KUKA KRL program: Dynamic_Mov.src

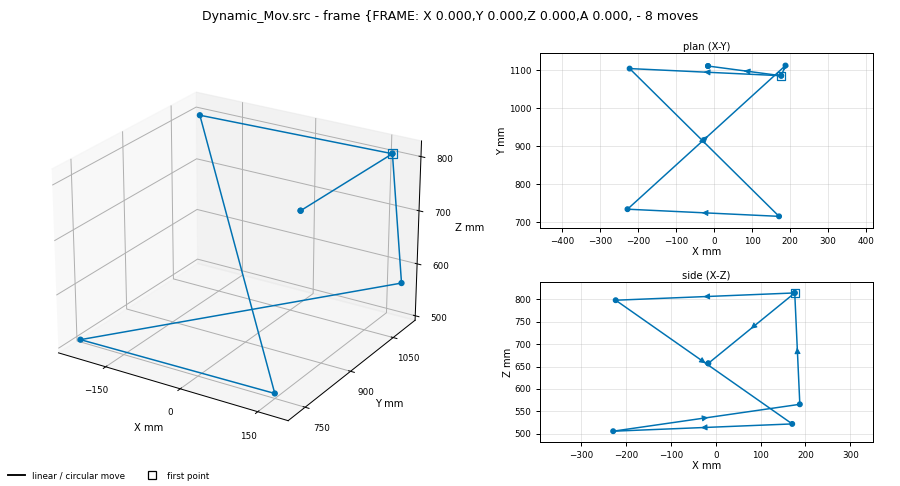
[picture p0: tool path of Dynamic_Mov.src in frame {FRAME: X 0.000,Y 0.000,Z 0.000,A 0.000,, 8 of 9 moves have a stored position in this frame; points joined in program order, loops and branches not executed]
&ACCESS RVP
&REL 1
&PARAM TEMPLATE = C:\KRC\Roboter\Template\vorgabe
&PARAM EDITMASK = *
DEF Kuka_Relative_Mo ( )
EXT BAS (BAS_COMMAND :IN,REAL :IN )


; GLOBAL INTERRUPT DECL 3 WHEN $STOPMESS==TRUE DO IR_STOPM ( )
; INTERRUPT ON 3

;FOLD Initialise and set default speed
BAS (#INITMOV,0)
BAS (#VEL_PTP,100)
BAS (#ACC_PTP,20)
$VEL.CP=0.2
BAS (#TOOL,0)
BAS (#BASE,0)
;ENDFOLD

;;FOLD STARTPOS
;$BWDSTART = FALSE
;PDAT_ACT = PDEFAULT
;BAS(#PTP_DAT)
;FDAT_ACT = {TOOL_NO 0,BASE_NO 0,IPO_FRAME #BASE}
;BAS(#FRAMES)
;;ENDFOLD

$ADVANCE = 5

;FOLD ---- Quickly skip BCO ----
; PTP $AXIS_ACT
;ENDFOLD

;FOLD ---- GO HOME ----
; PTP {A1 0.000, A2 -90.000, A3 90.000, A4 0.000, A5 0.000, A6 0.000, E1 0, E2 0, E3 0, E4 0, E5 0, E6 0}
;ENDFOLD


; Program generated by RoboDK v5.6.0 for KUKA KR 16 2 on 31/10/2023 10:24:52
; ---- Setting reference (Base) ----
$BASE = {FRAME: X 0.000,Y 0.000,Z 0.000,A 0.000,B 0.000,C 0.000}
; --------------------------
; ---- Setting tool (TCP) ----
; TOOL_DATA[1] = {FRAME: X 0.000,Y 0.000,Z 10.000,A 0.000,B 0.000,C 0.000}
$TOOL = {FRAME: X 0.000,Y 0.000,Z 10.000,A 0.000,B 0.000,C 0.000}
; $TOOL = TOOL_DATA[1]
; --------------------------
PTP {A1 -91.44,A2 -55.82,A3 116.05,A4 -4.21,A5 -66.58,A6 4.44}
; ---- Setting reference (Base) ----
$BASE = {FRAME: X 0.000,Y 0.000,Z 0.000,A 0.000,B 0.000,C 0.000}
; --------------------------
; ---- Setting tool (TCP) ----
$TOOL = {FRAME: X 0.000,Y 0.000,Z 10.000,A 0.000,B 0.000,C 0.000}
; --------------------------
LIN {X 176.195,Y 1085.310,Z 814.055,A 67.080,B 83.301,C -20.346}
; ---- Setting reference (Base) ----
$BASE = {FRAME: X 0.000,Y 0.000,Z 0.000,A 0.000,B 0.000,C 0.000}
; --------------------------
; ---- Setting tool (TCP) ----
$TOOL = {FRAME: X 0.000,Y 0.000,Z 10.000,A 0.000,B 0.000,C 0.000}
; --------------------------
LIN {X -223.032,Y 1104.150,Z 797.831,A 67.080,B 83.301,C -20.346}
; ---- Setting reference (Base) ----
$BASE = {FRAME: X 0.000,Y 0.000,Z 0.000,A 0.000,B 0.000,C 0.000}
; --------------------------
; ---- Setting tool (TCP) ----
$TOOL = {FRAME: X 0.000,Y 0.000,Z 10.000,A 0.000,B 0.000,C 0.000}
; --------------------------
LIN {X 170.586,Y 714.937,Z 522.011,A 67.080,B 83.301,C -20.346}
; ---- Setting reference (Base) ----
$BASE = {FRAME: X 0.000,Y 0.000,Z 0.000,A 0.000,B 0.000,C 0.000}
; --------------------------
; ---- Setting tool (TCP) ----
$TOOL = {FRAME: X 0.000,Y 0.000,Z 10.000,A 0.000,B 0.000,C 0.000}
; --------------------------
LIN {X -228.641,Y 733.776,Z 505.788,A 67.080,B 83.301,C -20.346}
; ---- Setting reference (Base) ----
$BASE = {FRAME: X 0.000,Y 0.000,Z 0.000,A 0.000,B 0.000,C 0.000}
; --------------------------
; ---- Setting tool (TCP) ----
$TOOL = {FRAME: X 0.000,Y 0.000,Z 10.000,A 0.000,B 0.000,C 0.000}
; --------------------------
LIN {X 187.552,Y 1112.180,Z 565.762,A 67.080,B 83.301,C -20.346}
; ---- Setting reference (Base) ----
$BASE = {FRAME: X 0.000,Y 0.000,Z 0.000,A 0.000,B 0.000,C 0.000}
; --------------------------
; ---- Setting tool (TCP) ----
$TOOL = {FRAME: X 0.000,Y 0.000,Z 10.000,A 0.000,B 0.000,C 0.000}
; --------------------------
LIN {X 176.195,Y 1085.310,Z 814.055,A 67.080,B 83.301,C -20.346}
; ---- Setting reference (Base) ----
$BASE = {FRAME: X 0.000,Y 0.000,Z 0.000,A 0.000,B 0.000,C 0.000}
; --------------------------
; ---- Setting tool (TCP) ----
$TOOL = {FRAME: X 0.000,Y 0.000,Z 10.000,A 0.000,B 0.000,C 0.000}
; --------------------------
LIN {X -16.604,Y 1110.850,Z 656.967,A 67.080,B 83.301,C -20.346}
; ---- Setting reference (Base) ----
$BASE = {FRAME: X 0.000,Y 0.000,Z 0.000,A 0.000,B 0.000,C 0.000}
; --------------------------
; ---- Setting tool (TCP) ----
$TOOL = {FRAME: X 0.000,Y 0.000,Z 10.000,A 0.000,B 0.000,C 0.000}
; --------------------------
LIN {X -16.604,Y 1110.850,Z 656.967,A 67.080,B 83.301,C -20.346}
END
